TYPE ST_MotorParameters :
	
STRUCT
	
fMinSpeed : REAL;
fMaxSpeed : REAL;

END_STRUCT

END_TYPE

(* stored: Version 1.1.0.1, ProductVersion 3.1.4024.12
   DUT ST_MotorParameters: Id {c347b47c-25f7-4f13-9460-a26b971f00e7} *)
